FUNCTION_BLOCK ValveControlledCylinder
VAR_INPUT
	ReturnPressure : LREAL;
	SupplyPressure : LREAL;
	par : ST_pValveControlledCylinder;
END_VAR
VAR_OUTPUT
END_VAR
VAR

//Pressure pA
fbPressureGradient_pA : PressureGradient;
PressurepA : LREAL;

//Pressure pB
fbPressureGradient_pB : PressureGradient;
PressurepB : LREAL;

//OrificeEquation QA and QB
fbOrificeEquationQ_P_A : OrificeEquation;
fbOrificeEquationQ_B_R : OrificeEquation;
fbOrificeEquationQ_P_B : OrificeEquation;
fbOrificeEquationQ_A_R : OrificeEquation;	
FlowQ_P_A : LREAL;
FlowQ_B_R : LREAL;	
FlowQ_P_B : LREAL;
FlowQ_A_R : LREAL;
FlowQA : LREAL;
FlowQB : LREAL;

//HydraulicCylinder
fbHydraulicCylinder : HydraulicCylinder;

xPos : LREAL;
ValveOpeningControl : LREAL := 0.0;

fbBulkModulus : BulkModulus;

END_VAR

//Pressure Gradient pA and Pressure pA
fbPressureGradient_pA(
	TotalVolume := par.VA0 + (fbHydraulicCylinder.PistonPosition * fbHydraulicCylinder.Aa),
	BulkModulus := fbBulkModulus.BulkModulus,
	FlowrateIn := FlowQA,
	FlowrateOut := (fbHydraulicCylinder.PistonVelocity * fbHydraulicCylinder.Aa),
	p0 := par.pA0,
	param := par,
	Pressure => PressurepA		//Pressure
	);

//Pressure Gradient pB and Pressure pB
fbPressureGradient_pB(
	TotalVolume := par.VB0 + ((par.xMax - fbHydraulicCylinder.PistonPosition) * fbHydraulicCylinder.Ab),
	BulkModulus := fbBulkModulus.BulkModulus,
	FlowrateIn := (fbHydraulicCylinder.PistonVelocity * fbHydraulicCylinder.Ab),
	FlowrateOut := FlowQB,
	p0 := par.pB0,
	param := par,
	Pressure => PressurepB		//Pressure
	);

fbOrificeEquationQ_P_A(
	PressureOut := PressurepA, 			//Found value from old simulink project, this one goes to the tank i guess
	PressureIn := SupplyPressure,	
	ValveOpening := ValveOpeningControl,	
	param := par,
	OrificeFlow => FlowQ_P_A
	);
	
fbOrificeEquationQ_A_R(
	PressureOut := ReturnPressure, 			//Found value from old simulink project, this one goes to the tank i guess
	PressureIn :=  PressurepA,	
	ValveOpening := ValveOpeningControl,	
	param := par,
	OrificeFlow => FlowQ_A_R
	);


	
fbOrificeEquationQ_B_R(
	PressureOut := ReturnPressure, 			//Found value from old simulink project, this one goes to the tank i guess
	PressureIn := PressurepB,			
	ValveOpening := ValveOpeningControl,
	param := par,
	OrificeFlow => FlowQ_B_R
	);
	
fbOrificeEquationQ_P_B(
	PressureOut := PressurepB, 			//Found value from old simulink project, this one goes to the tank i guess
	PressureIn := SupplyPressure,			
	ValveOpening := ValveOpeningControl,
	param := par,
	OrificeFlow => FlowQ_P_B
	);	

IF ValveOpeningControl > 0 THEN
	FlowQA := FlowQ_P_A;		
	FlowQB := FlowQ_B_R;
ELSIF ValveOpeningControl < 0 THEN
	FlowQA := FlowQ_A_R;		
	FlowQB := FlowQ_P_B;
ELSE
	FlowQA := 0.0;		
	FlowQB := 0.0;	
END_IF

	
//Hydraulic Cylinder 1
fbHydraulicCylinder(
	PressureBoreSide := PressurepA,
	PressureRodSide := PressurepB,
	PistonPosition => xPos,
	param := Param.pMainJibCylinder
	);

END_FUNCTION_BLOCK

(* stored: Version 1.1.0.1, ProductVersion 3.1.4024.9
   POU ValveControlledCylinder: Id {c1915dd1-7c80-44ad-a4db-c25faf141489}, SpecialFunc None *)
